(* PLC project Unnamed, Unknown Unnamed 1 *)
(* stored: creationDateTime 2025-09-23T07:17:21, modificationDateTime 2025-09-27T15:46:03 *)

PROGRAM test_program
  VAR
    SWITCH_0 : BOOL;
    LED_0 : BOOL;
  END_VAR

(* LD diagram, written out as Structured Text *)
END_PROGRAM

CONFIGURATION Config0
  RESOURCE Res0 ON PLC
  END_RESOURCE
END_CONFIGURATION
